RoboDK station: RBT23CS084-mdm-practical-object_sorting.rdk

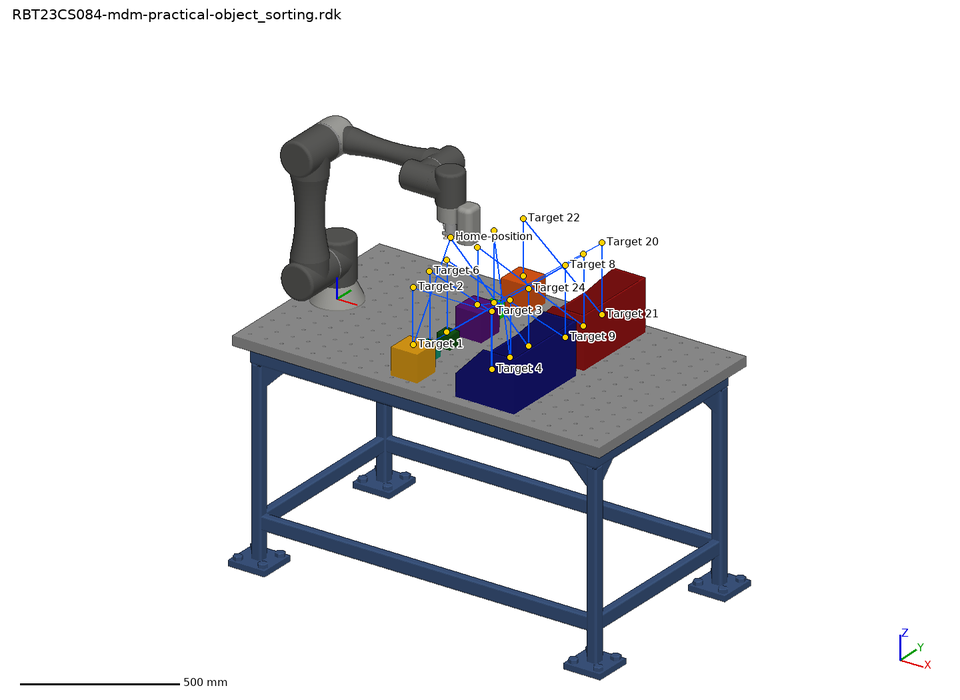
[picture v0: the station drawn from its stored meshes, robots at their saved joint values, targets as dots, program paths as lines]
Station RBT23CS084-mdm-practical-object_sorting (saved by RoboDK 5.9.2). Poses are relative to the parent item; angles as X-Y-Z fixed-axis rotations.
  - frame TM5-900 Base at (0, 0, 0) mm
    - robot TM5-900: 6 axes, payload 4 kg, reach 900 mm, repeatability 0.1 mm, weight 30 kg
        modified DH rows (alpha deg, a mm, theta deg, d mm): 0, 0, 0, 145.2; 90, 0, 90, 0; 0, 429, 0, 0; 0, 411, -90, 122.3; -90, 0, 0, 106.5; 90, 0, 180, 114.15
        joint limits [-360, -180, -155, -180, -180, -270] to [360, 180, 155, 180, 180, 270]; home [0, 0, 90, -90, 90, 0]; saved at [0, 0.016, 88.59, 1.394, 90, 0]
      - tool SMC ZXP7A01-ZP25C-X1 Vacuum Gripper, TCP at (0, 0, 62.5) mm, size 44 x 53.4 x 64 mm
    - target Home-position (Cartesian target) at (517.5, -122.3, 407.55) mm, rotated rx 180 ry 0 rz 90 deg; joints [0, 0.016, 88.59, 1.394, 90, 0] of TM5-900
    - target Target 1 (Cartesian target) at (500, -300, 100) mm, rotated rx 180 ry 0 rz 90 deg; joints [-18.856, 20.913, 110.022, -40.935, 90, -18.856] of TM5-900
    - target Target 2 (Cartesian target) at (500, -300, 300) mm, rotated rx 180 ry 0 rz 90 deg; joints [-18.856, 8.479, 94.579, -13.058, 90, -18.856] of TM5-900
    - target Target 3 (Cartesian target) at (800, -300, 300) mm, rotated rx 180 ry 0 rz 90 deg; joints [-12.326, 50.826, 30.715, 8.459, 90, -12.326] of TM5-900
    - target Target 4 (Cartesian target) at (800, -300, 100) mm, rotated rx 180 ry 0 rz 90 deg; joints [-12.326, 53.866, 53.332, -17.198, 90, -12.326] of TM5-900
    - target Target 5 (Cartesian target) at (800, -300, 300) mm, rotated rx 180 ry 0 rz 90 deg; joints [-12.326, 50.826, 30.715, 8.459, 90, -12.326] of TM5-900
    - target Target 6 (Cartesian target) at (475, -175, 300) mm, rotated rx 180 ry 0 rz 90 deg; joints [-6.244, -1.95, 105.645, -13.694, 90, -6.244] of TM5-900
    - target Target 7 (Cartesian target) at (475, -175, 50) mm, rotated rx 180 ry 0 rz 90 deg; joints [-6.244, 18.254, 124.222, -52.476, 90, -6.244] of TM5-900
    - target Target 8 (Cartesian target) at (800, 100, 300) mm, rotated rx 180 ry 0 rz 90 deg; joints [15.85, 40.645, 48.526, 0.828, 90, 15.85] of TM5-900
    - target Target 9 (Cartesian target) at (800, 100, 50) mm, rotated rx 180 ry 0 rz 90 deg; joints [15.85, 49.949, 68.312, -28.261, 90, 15.85] of TM5-900
    - target Target 10 (Cartesian target) at (475, -80, 300) mm, rotated rx 180 ry 0 rz 90 deg; joints [5.148, -5.392, 108.849, -13.458, 90, 5.148] of TM5-900
    - target Target 11 (Cartesian target) at (475, -80, 50) mm, rotated rx -180 ry 0 rz 90 deg; joints [5.148, 15.742, 128.01, -53.752, 90, 5.148] of TM5-900
    - target Target 12 (Cartesian target) at (800, 200, 300) mm, rotated rx 180 ry 0 rz 90 deg; joints [22.565, 44.124, 42.599, 3.277, 90, 22.565] of TM5-900
    - target Target 13 (Cartesian target) at (800, 200, 50) mm, rotated rx 180 ry 0 rz 90 deg; joints [22.565, 52.369, 63.68, -26.049, 90, 22.565] of TM5-900
    - target Target 14 (Cartesian target) at (500, 50, 300) mm, rotated rx 180 ry 0 rz 90 deg; joints [19.797, -2.467, 106.14, -13.673, 90, 19.797] of TM5-900
    - target Target 15 (Cartesian target) at (500, 50, 100) mm, rotated rx 180 ry 0 rz 90 deg; joints [19.797, 11.847, 122.72, -44.566, 90, 19.797] of TM5-900
    - target Target 16 (Cartesian target) at (800, -200, 300) mm, rotated rx 180 ry 0 rz 90 deg; joints [-5.507, 44.124, 42.599, 3.277, 90, -5.507] of TM5-900
    - target Target 17 (Cartesian target) at (800, -200, 100) mm, rotated rx 180 ry 0 rz 90 deg; joints [-5.507, 49.364, 61.733, -21.097, 90, -5.507] of TM5-900
    - target Target 18 (Cartesian target) at (475, 175, 300) mm, rotated rx 180 ry 0 rz 90 deg; joints [34.206, -1.95, 105.645, -13.694, 90, 34.206] of TM5-900
    - target Target 19 (Cartesian target) at (475, 175, 50) mm, rotated rx 180 ry 0 rz 90 deg; joints [34.206, 18.254, 124.222, -52.476, 90, 34.206] of TM5-900
    - target Target 20 (Cartesian target) at (800, 300, 300) mm, rotated rx 180 ry 0 rz 90 deg; joints [28.786, 50.826, 30.715, 8.459, 90, 28.786] of TM5-900
    - target Target 21 (Cartesian target) at (800, 300, 50) mm, rotated rx 180 ry 0 rz 90 deg; joints [28.786, 56.627, 55.459, -22.086, 90, 28.786] of TM5-900
    - target Target 22 (Cartesian target) at (500, 300, 300) mm, rotated rx 180 ry 0 rz 90 deg; joints [43.071, 8.479, 94.579, -13.058, 90, 43.071] of TM5-900
    - target Target 23 (Cartesian target) at (500, 300, 100) mm, rotated rx 180 ry 0 rz 90 deg; joints [43.071, 20.913, 110.022, -40.935, 90, 43.071] of TM5-900
    - target Target 24 (Cartesian target) at (800, -100, 300) mm, rotated rx 180 ry 0 rz 90 deg; joints [1.6, 40.645, 48.526, 0.828, 90, 1.6] of TM5-900
    - target Target 25 (Cartesian target) at (800, -100, 100) mm, rotated rx 180 ry 0 rz 90 deg; joints [1.6, 46.805, 66.438, -23.243, 90, 1.6] of TM5-900
    - target End-position (Cartesian target) at (517.5, -122.3, 407.55) mm, rotated rx 180 ry 0 rz 90 deg; joints [0, 0.016, 88.59, 1.394, 90, 0] of TM5-900
  - object Table 1400x800x800mm at (220, 0, 0) mm, size 1420 x 820 x 800 mm, geometry from Table-1400x800x800mm.sld
  - object Bin Blue at (700, -20, 0) mm, rotated rx 0 ry 0 rz 180 deg, size 225 x 337.5 x 191.2 mm, geometry from Bin-Blue.sld
  - object Bin Red at (700, 360, 0) mm, rotated rx 0 ry 0 rz 180 deg, size 225 x 337.5 x 191.2 mm, geometry from Bin-Red.sld
  - program Prog1 (41 instructions, listed below)
  - object Cube-large-3 at (450, 250, 0) mm, size 100 x 100 x 100 mm, geometry from Cube-100mm.sld
  - object Cube-small-3 at (450, 150, 0) mm, size 50 x 50 x 50 mm, geometry from Cube-50mm.sld
  - object Cube-large-2 at (450, 0, 0) mm, size 100 x 100 x 100 mm, geometry from Cube-100mm.sld
  - object Cube-small-2 at (450, -100, 0) mm, size 50 x 50 x 50 mm, geometry from Cube-50mm.sld
  - object Cube-small-1 at (450, -200, 0) mm, size 50 x 50 x 50 mm, geometry from Cube-50mm.sld
  - object Cube-large-1 at (450, -350, 0) mm, size 100 x 100 x 100 mm, geometry from Cube-100mm.sld
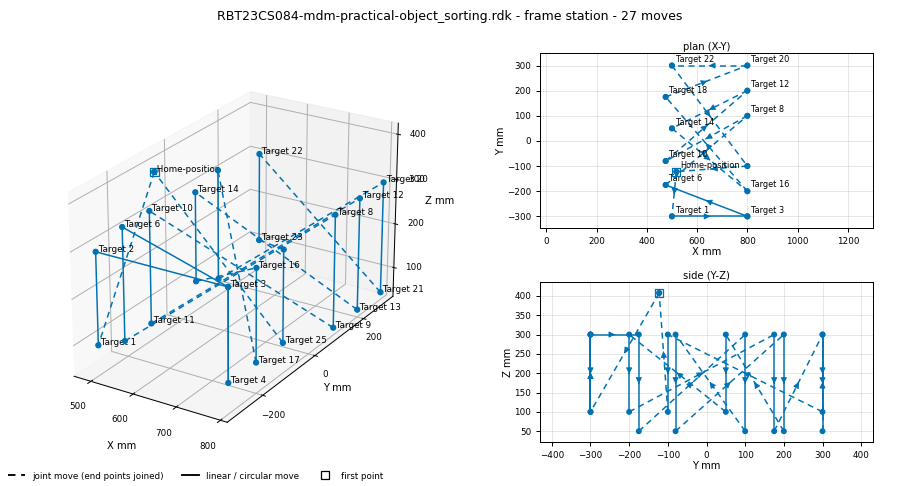
[picture p0: tool path of RBT23CS084-mdm-practical-object_sorting.rdk in frame station, 27 of 27 moves have a stored position in this frame; points joined in program order, loops and branches not executed]

--- program Prog1 (robot TM5-900) ---
  Set Ref.: TM5-900 Base
  Set Tool: SMC ZXP7A01-ZP25C-X1 Vacuum Gripper
  MoveJ (Home-position)
  MoveJ (Target 1)
  Attach to SMC ZXP7A01-ZP25C-X1 Vacuum Gripper
  MoveL (Target 2)
  MoveL (Target 3)
  MoveL (Target 4)
  Detach from SMC ZXP7A01-ZP25C-X1 Vacuum Gripper
  MoveL (Target 5)
  MoveL (Target 6)
  MoveL (Target 7)
  Attach to SMC ZXP7A01-ZP25C-X1 Vacuum Gripper
  MoveJ (Target 8)
  MoveL (Target 9)
  Detach from SMC ZXP7A01-ZP25C-X1 Vacuum Gripper
  MoveJ (Target 10)
  MoveL (Target 11)
  Attach to SMC ZXP7A01-ZP25C-X1 Vacuum Gripper
  MoveJ (Target 12)
  MoveL (Target 13)
  Detach from SMC ZXP7A01-ZP25C-X1 Vacuum Gripper
  MoveJ (Target 14)
  MoveL (Target 15)
  Attach to SMC ZXP7A01-ZP25C-X1 Vacuum Gripper
  MoveJ (Target 16)
  MoveL (Target 17)
  Detach from SMC ZXP7A01-ZP25C-X1 Vacuum Gripper
  MoveJ (Target 18)
  MoveL (Target 19)
  Attach to SMC ZXP7A01-ZP25C-X1 Vacuum Gripper
  MoveJ (Target 20)
  MoveL (Target 21)
  Detach from SMC ZXP7A01-ZP25C-X1 Vacuum Gripper
  MoveJ (Target 22)
  MoveL (Target 23)
  Attach to SMC ZXP7A01-ZP25C-X1 Vacuum Gripper
  MoveJ (Target 24)
  MoveL (Target 25)
  Detach from SMC ZXP7A01-ZP25C-X1 Vacuum Gripper
  MoveJ (End-position)
